// TIA Portal project "btvn2" (V16)

(* hardware
DEVICE "S7300/ET200M station_1"  S7-300 station
   slot 0: "Rail_0"  Rail  6ES7 390-1***0-0AA0
   slot 2: "PLC"  CPU 314C-2 PN/DP  6ES7 314-6EH04-0AB0  V3.3
      slot 2: "PROFINET interface_1"  PN-IO
         slot 1: "Port_1"  Port
         slot 2: "Port_2"  Port
      slot 5: "DI 24/DO 16_1"  DI24/DO16
      slot 6: "AI 5/AO 2_1"  AI5/AO2
      slot 7: "Count_1"  Counter
      slot 8: "Positioning_1"  Positioning
DEVICE "HMI"  TP900 Comfort
   slot 0: "HMI"  TP900 Comfort  6AV2 124-0JC01-0AX0  16.0.0.0
   slot 1: "HMI_RT_1"  TP900 Comfort  6AV2 124-0JC01-0AX0  16.0.0.0
   slot 5: "HMI.IE_CP_1"  PROFINET Interface  16.0.0.0
      slot 1: "PROFINET Interface_1"  PROFINET Interface
         slot 1: "Port_1"  Port
         slot 2: "Port_2"  Port
   slot 7: "HMI.MPI/DP_CP_1"  MPI/DP Interface  16.0.0.0
*)

// ===== PLC "PLC"  CPU 314C-2 PN/DP =====

VAR_GLOBAL   // PLC tag table "Default tag table"
   "S1" AT %M0.0 : Bool;
   "S2" AT %M0.1 : Bool;
   "S3" AT %M0.2 : Bool;
   "S4" AT %M0.3 : Bool;
   "R_do" AT %Q0.4 : Bool;
   "Y_vang" AT %Q0.5 : Bool;
   "G_XANH" AT %Q0.6 : Bool;
   "Q1" AT %Q0.0 : Bool;
   "Q2" AT %Q0.1 : Bool;
   "Q3" AT %Q0.2 : Bool;
   "Q4" AT %Q0.3 : Bool;
   "Tag_1" AT %Q1.0 : Bool;
   "Tag_2" AT %Q1.1 : Bool;
   "Tag_3" AT %Q1.2 : Bool;
   "Tag_4" AT %Q1.3 : Bool;
   "Tag_5" AT %M1.0 : Bool;
   "Tag_6" AT %M1.1 : Bool;
   "Tag_7" AT %M1.2 : Bool;
   "Tag_8" AT %M1.3 : Bool;
   "Tag_9" AT %M1.4 : Bool;
   "Tag_10" AT %M1.5 : Bool;
   "Tag_11" AT %M1.6 : Bool;
   "Tag_12" AT %M1.7 : Bool;
   "Tag_13" AT %M2.0 : Bool;
   "Tag_14" AT %M2.1 : Bool;
   "Tag_15" AT %M2.2 : Bool;
END_VAR

ORGANIZATION_BLOCK "Main"   // OB1, LAD
TITLE = "Main Program Sweep (Cycle)"
{ S7_Optimized_Access := 'FALSE' }
VERSION : 0.1
   VAR_TEMP
      OB1_EV_CLASS : Byte;   // Bits 0-3 = 1 (Coming event), Bits 4-7 = 1 (Event class 1)
      OB1_SCAN_1 : Byte;   // 1 (Cold restart scan 1 of OB 1), 3 (Scan 2-n of OB 1)
      OB1_PRIORITY : Byte;   // Priority of OB Execution
      OB1_OB_NUMBR : Byte;   // 1 (Organization block 1, OB1)
      OB1_RESERVED_1 : Byte;   // Reserved for system
      OB1_RESERVED_2 : Byte;   // Reserved for system
      OB1_PREV_CYCLE : Int;   // Cycle time of previous OB1 scan (milliseconds)
      OB1_MIN_CYCLE : Int;   // Minimum cycle time of OB1 (milliseconds)
      OB1_MAX_CYCLE : Int;   // Maximum cycle time of OB1 (milliseconds)
      OB1_DATE_TIME : Date_And_Time;   // Date and time OB1 started
   END_VAR
   VAR_TEMP   // added for the SCL form of the ladder/FBD networks
      _w1 : Bool;
   END_VAR
BEGIN

REGION Network 1
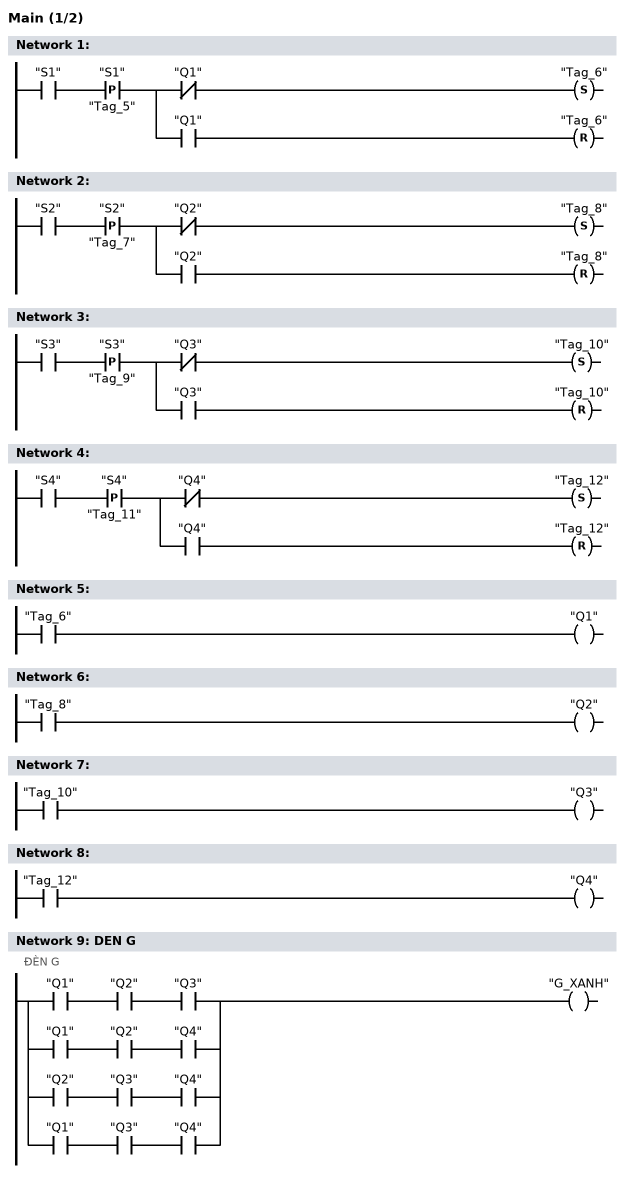
   RUNG wire#powerrail
      Contact( "S1" )
      P_Contact(operand := "S1", bit := "Tag_5")
      wire#w1
      I_Contact( "Q1" )
      S_Coil( "Tag_6" )
   END_RUNG
   RUNG wire#w1
      Contact( "Q1" )
      R_Coil( "Tag_6" )
   END_RUNG
   // the same network as SCL:
   #_w1 := "S1" AND "S1" AND NOT "Tag_5";   // rising edge of "S1"
   "Tag_5" := "S1";
   IF #_w1 AND NOT "Q1" THEN "Tag_6" := TRUE; END_IF;
   IF #_w1 AND "Q1" THEN "Tag_6" := FALSE; END_IF;
END_REGION

REGION Network 2
   RUNG wire#powerrail
      Contact( "S2" )
      P_Contact(operand := "S2", bit := "Tag_7")
      wire#w1
      I_Contact( "Q2" )
      S_Coil( "Tag_8" )
   END_RUNG
   RUNG wire#w1
      Contact( "Q2" )
      R_Coil( "Tag_8" )
   END_RUNG
   // the same network as SCL:
   #_w1 := "S2" AND "S2" AND NOT "Tag_7";   // rising edge of "S2"
   "Tag_7" := "S2";
   IF #_w1 AND NOT "Q2" THEN "Tag_8" := TRUE; END_IF;
   IF #_w1 AND "Q2" THEN "Tag_8" := FALSE; END_IF;
END_REGION

REGION Network 3
   RUNG wire#powerrail
      Contact( "S3" )
      P_Contact(operand := "S3", bit := "Tag_9")
      wire#w1
      I_Contact( "Q3" )
      S_Coil( "Tag_10" )
   END_RUNG
   RUNG wire#w1
      Contact( "Q3" )
      R_Coil( "Tag_10" )
   END_RUNG
   // the same network as SCL:
   #_w1 := "S3" AND "S3" AND NOT "Tag_9";   // rising edge of "S3"
   "Tag_9" := "S3";
   IF #_w1 AND NOT "Q3" THEN "Tag_10" := TRUE; END_IF;
   IF #_w1 AND "Q3" THEN "Tag_10" := FALSE; END_IF;
END_REGION

REGION Network 4
   RUNG wire#powerrail
      Contact( "S4" )
      P_Contact(operand := "S4", bit := "Tag_11")
      wire#w1
      I_Contact( "Q4" )
      S_Coil( "Tag_12" )
   END_RUNG
   RUNG wire#w1
      Contact( "Q4" )
      R_Coil( "Tag_12" )
   END_RUNG
   // the same network as SCL:
   #_w1 := "S4" AND "S4" AND NOT "Tag_11";   // rising edge of "S4"
   "Tag_11" := "S4";
   IF #_w1 AND NOT "Q4" THEN "Tag_12" := TRUE; END_IF;
   IF #_w1 AND "Q4" THEN "Tag_12" := FALSE; END_IF;
END_REGION

REGION Network 5
   RUNG wire#powerrail
      Contact( "Tag_6" )
      Coil( "Q1" )
   END_RUNG
   // the same network as SCL:
   "Q1" := "Tag_6";
END_REGION

REGION Network 6
   RUNG wire#powerrail
      Contact( "Tag_8" )
      Coil( "Q2" )
   END_RUNG
   // the same network as SCL:
   "Q2" := "Tag_8";
END_REGION

REGION Network 7
   RUNG wire#powerrail
      Contact( "Tag_10" )
      Coil( "Q3" )
   END_RUNG
   // the same network as SCL:
   "Q3" := "Tag_10";
END_REGION

REGION Network 8
   RUNG wire#powerrail
      Contact( "Tag_12" )
      Coil( "Q4" )
   END_RUNG
   // the same network as SCL:
   "Q4" := "Tag_12";
END_REGION

REGION Network 9: DEN G
   // ĐÈN G
   RUNG wire#powerrail
      Contact( "Q1" )
      Contact( "Q2" )
      Contact( "Q3" )
      wire#w1
      Coil( "G_XANH" )
   END_RUNG
   RUNG wire#powerrail
      Contact( "Q1" )
      Contact( "Q2" )
      Contact( "Q4" )
   END_RUNG wire#w1
   RUNG wire#powerrail
      Contact( "Q2" )
      Contact( "Q3" )
      Contact( "Q4" )
   END_RUNG wire#w1
   RUNG wire#powerrail
      Contact( "Q1" )
      Contact( "Q3" )
      Contact( "Q4" )
   END_RUNG wire#w1
   // the same network as SCL:
   "G_XANH" := ("Q1" AND "Q2" AND "Q3") OR ("Q1" AND "Q2" AND "Q4") OR ("Q2" AND "Q3" AND "Q4") OR ("Q1" AND "Q3" AND "Q4");
END_REGION

REGION Network 10: DEN Y
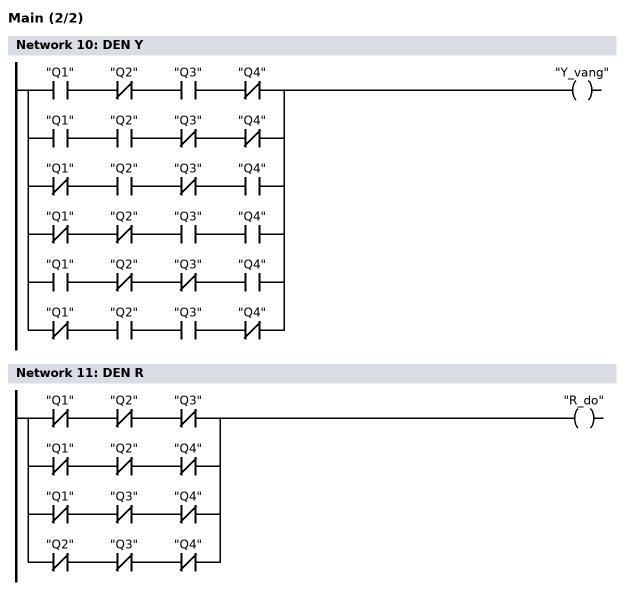
   RUNG wire#powerrail
      Contact( "Q1" )
      I_Contact( "Q2" )
      Contact( "Q3" )
      I_Contact( "Q4" )
      wire#w1
      Coil( "Y_vang" )
   END_RUNG
   RUNG wire#powerrail
      Contact( "Q1" )
      Contact( "Q2" )
      I_Contact( "Q3" )
      I_Contact( "Q4" )
   END_RUNG wire#w1
   RUNG wire#powerrail
      I_Contact( "Q1" )
      Contact( "Q2" )
      I_Contact( "Q3" )
      Contact( "Q4" )
   END_RUNG wire#w1
   RUNG wire#powerrail
      I_Contact( "Q1" )
      I_Contact( "Q2" )
      Contact( "Q3" )
      Contact( "Q4" )
   END_RUNG wire#w1
   RUNG wire#powerrail
      Contact( "Q1" )
      I_Contact( "Q2" )
      I_Contact( "Q3" )
      Contact( "Q4" )
   END_RUNG wire#w1
   RUNG wire#powerrail
      I_Contact( "Q1" )
      Contact( "Q2" )
      Contact( "Q3" )
      I_Contact( "Q4" )
   END_RUNG wire#w1
   // the same network as SCL:
   "Y_vang" := ("Q1" AND NOT "Q2" AND "Q3" AND NOT "Q4") OR ("Q1" AND "Q2" AND NOT "Q3" AND NOT "Q4") OR (NOT "Q1" AND "Q2" AND NOT "Q3" AND "Q4") OR (NOT "Q1" AND NOT "Q2" AND "Q3" AND "Q4") OR ("Q1" AND NOT "Q2" AND NOT "Q3" AND "Q4") OR (NOT "Q1" AND "Q2" AND "Q3" AND NOT "Q4");
END_REGION

REGION Network 11: DEN R
   RUNG wire#powerrail
      I_Contact( "Q1" )
      I_Contact( "Q2" )
      I_Contact( "Q3" )
      wire#w1
      Coil( "R_do" )
   END_RUNG
   RUNG wire#powerrail
      I_Contact( "Q1" )
      I_Contact( "Q2" )
      I_Contact( "Q4" )
   END_RUNG wire#w1
   RUNG wire#powerrail
      I_Contact( "Q1" )
      I_Contact( "Q3" )
      I_Contact( "Q4" )
   END_RUNG wire#w1
   RUNG wire#powerrail
      I_Contact( "Q2" )
      I_Contact( "Q3" )
      I_Contact( "Q4" )
   END_RUNG wire#w1
   // the same network as SCL:
   "R_do" := (NOT "Q1" AND NOT "Q2" AND NOT "Q3") OR (NOT "Q1" AND NOT "Q2" AND NOT "Q4") OR (NOT "Q1" AND NOT "Q3" AND NOT "Q4") OR (NOT "Q2" AND NOT "Q3" AND NOT "Q4");
END_REGION
END_ORGANIZATION_BLOCK

(* ===== HMI "HMI_RT_1" =====
system functions are stored by id; their names below are inferred from use
connection "HMI_Connection_1": ETHERNET, SIMATIC S7 300/400 MPI

HMI tags "Default tag table"
   "S1" : Bool = PLC S1 AT %M0.0, 1 s
   "S2" : Bool = PLC S2 AT %M0.1, 1 s
   "S3" : Bool = PLC S3 AT %M0.2, 1 s
   "S4" : Bool = PLC S4 AT %M0.3, 1 s
   "R_do" : Bool = PLC R_do AT %Q0.4, 1 s
   "Y_vang" : Bool = PLC Y_vang AT %Q0.5, 1 s
   "G_XANH" : Bool = PLC G_XANH AT %Q0.6, 1 s
   "Q1" : Bool = PLC Q1 AT %Q0.0, 1 s
   "Q2" : Bool = PLC Q2 AT %Q0.1, 1 s
   "Q3" : Bool = PLC Q3 AT %Q0.2, 1 s
   "Q4" : Bool = PLC Q4 AT %Q0.3, 1 s

screen "Main" 800x480
   TextField "Text field_1" at 74,58 size 82x20; Text 'Điều khiển'
   Button "Button_1" at 60,91 size 96x32; TextOff 'S1'
      Appearance <- "S1"
      on Press: SetBit("S1")
      on Release: ResetBit("S1")
   Button "Button_2" at 60,137 size 96x32; TextOff 'S2'
      Appearance <- "S2"
      on Press: SetBit("S2")
      on Release: ResetBit("S2")
   Button "Button_3" at 60,181 size 96x32; TextOff 'S3'
      Appearance <- "S3"
      on Release: ResetBit("S3")
      on Press: SetBit("S3")
   Button "Button_4" at 60,225 size 96x32; TextOff 'S4'
      Appearance <- "S4"
      on Press: SetBit("S4")
      on Release: ResetBit("S4")
   TextField "Text field_2" at 188,58 size 40x20; Text 'Quạt'
   Circle "Circle_1" at 188,86 size 37x37
      Appearance <- "Q1"
   Circle "Circle_2" at 188,176 size 37x37
      Appearance <- "Q3"
   Circle "Circle_3" at 188,132 size 37x37
      Appearance <- "Q2"
   Circle "Circle_4" at 188,225 size 37x37
      Appearance <- "Q4"
   TextField "Text field_3" at 199,91 size 14x20; Text '1'
   TextField "Text field_4" at 199,137 size 14x20; Text '2'
   TextField "Text field_5" at 199,181 size 14x20; Text '3'
   TextField "Text field_6" at 199,231 size 14x20; Text '4'
   TextField "Text field_7" at 541,23 size 34x20; Text 'Đèn'
   Circle "Circle_5" at 407,74 size 37x37
      Appearance <- "R_do"
   Circle "Circle_6" at 541,74 size 37x37
      Appearance <- "Y_vang"
   Circle "Circle_7" at 675,74 size 37x37
      Appearance <- "G_XANH"
   TextField "Text field_8" at 410,58 size 25x20; Text 'Đỏ'
   TextField "Text field_9" at 541,58 size 42x20; Text 'Vàng'
   TextField "Text field_10" at 672,58 size 42x20; Text 'Xanh'
*)